FUNCTION_BLOCK Test_GetTestReturnsCorrectTest EXTENDS T_UnitTestBase
VAR
	List : T_ListOfTests(Capacity := 10,TestGroupName := 'Unit Tests');
	Test1 : T_UnitTestBase(List);
	Test2 : T_UnitTestBase(List);
	Test3 : T_UnitTestBase(List);
	Test4 : T_UnitTestBase(List);
	
	Result : I_UnitTest;
END_VAR

Result := List.GetTest(2);


Assertion.AssertEquals_STRING(Expected     := 'Test3',
                            Actual       := Result.TestName,
                            VariableName := 'Result.TestName');
							
CheckAssertion(NextState := 0);

END_FUNCTION_BLOCK

(* stored: Version 1.1.0.1, ProductVersion 3.1.4024.11
   POU Test_GetTestReturnsCorrectTest: Id {c9448291-0ac7-4baf-aa2f-b789133876a8}, SpecialFunc None *)
